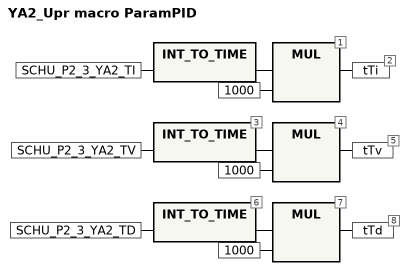
[picture p516: YA2_Upr macro ParamPID (CFC)]
_CFC_ (* Continuous Function Chart, elements in execution order *)
#0 TON_SCHU_P2_3_P1_DI4_RUN:TON(IN: SCHU_P2_3_P1_DI4_RUN, PT: T#10s)
#1 AND(SCHU_P2_3_UST_RE_RABOTA, #0.Q)
#2 reg1 <= #1
#3 AND(NOT SCHU_P2_3_UST_RE_RABOTA, #0.Q, NOT SCHU_P2_3_UST_RE_PROGREV)
#4 reg2 <= #3
#5 AND(reg1, SCHU_P2_3_UE1_T_DOST)
#6 AND(reg2, SCHU_P2_3_TE2_DOST)
#7 OR(#5, #6)
#8 YA2_DOST <= #7
#9 MACRO ParamPID()
	#10 INT_TO_TIME(SCHU_P2_3_YA2_TI)
	#11 MUL(#10, 1000)
	#12 tTi <= #11
	#13 INT_TO_TIME(SCHU_P2_3_YA2_TV)
	#14 MUL(#13, 1000)
	#15 tTv <= #14
	#16 INT_TO_TIME(SCHU_P2_3_YA2_TD)
	#17 MUL(#16, 1000)
	#18 tTd <= #17
END_MACRO
#19 SUB(SCHU_P2_3_UE2_T_UST, SCHU_P2_3_TE2_VN)
#20 EPS2 <= #19
#21 SUB(SCHU_P2_3_UE2_T_UST, SCHU_P2_3_UE1_T_VN)
#22 EPS1 <= #21
#23 SEL(reg1, SCHU_P2_3_TE2_UST, SCHU_P2_3_UE1_T_UST)
#24 >(EPS1, EPS2)
#25 AND(reg1, #24)
#26 SEL(#25, SCHU_P2_3_TE2_VN, SCHU_P2_3_UE1_T_VN)
#27 OR(reg1, reg2)
#28 AND(#27, YA2_DOST)
#29 SEL(#28, 0, #23)
#30 SEL(#28, 0, #26)
#31 AND(#28, SCHU_P2_3_SA4_DI3_A)
#32 SCHU_P2_3_YA2_AUTO <= #31
#33 AND(NOT SCHU_P2_3_TE1_B_UST_MYAG_REG, SCHU_P2_3_UST_RE_PROGREV)
#34 OR(Z_ZAM_SR, #33)
#35 AND(#31, NOT #34)
#36 AND(#35, NOT SCHU_P2_3_Z_GVS1_OTKAZ)
#37 YA2_REG_POL <= #36
#38 SEL(#36, eHVACCtrlMode_Manual, eHVACCtrlMode_Auto)
#39 SEL(NOT SCHU_P2_3_P1_DI4_RUN, SCHU_P2_3_YA2_UP_VN, rYMin)
#40 SEL(SCHU_P2_3_UST_RE_PROGREV, #39, 50)
#41 SEL(#34, #40, 100)
#42 SEL(SCHU_P2_3_SA4_DI3_A, SCHU_P2_3_YA2_UP_VN, #41)
#43 SEL(SCHU_P2_3_Z_GVS1_OTKAZ, #42, 0)
#44 YA2_PID:FB_HVACPIDCtrl(eHVACDataSecurityType_Idle, FALSE, TRUE, #29, #30, tTaskCycleTime, tTaskCycleTime, #38, #43, SCHU_P2_3_YA2_UP_VN, FALSE, SCHU_P2_3_SB, deadRange, direction, SCHU_P2_3_YA2_KP, tTi, tTv, tTd, rYMin, rYMax)
#45 SCHU_P2_3_YA2_RASSOG <= #44.out 2
#46 YA2_OTKAZ <= #44.out 8
#47 SEL(SCHU_P2_3_SA4_DI3_A, 0, #44.out 1)
#48 SCHU_P2_3_YA2_ZAD_VN <= #47
#49 SUB(#47, SCHU_P2_3_YA2_UP_VN)
#50 SCHU_P2_3_YA2_RASSOG_POL <= #49
#51 SEL(SCHU_P2_3_UST_ZIMA, 0, SCHU_P2_3_YA2_UP_MIN)
#52 rYMin <= #51
_END_CFC_
END_PROGRAM

(* POU IM/YA3_Upr, CFC *)
PROGRAM YA3_Upr
VAR
	YA3_PID: FB_HVACPIDCtrl;

	deadRange: REAL := 0.1;
	direction: BOOL := TRUE;
	tTi: TIME;
	tTv: TIME;
	tTd: TIME;

	rYMin: REAL := 0;
	rYMax: REAL := 100;
END_VAR
